(* Logix 5000 project; controller TWO_SRC_TEST vendor 1 type 14 code 54 rev 19.11; software revision 19.01 *)
// Two sources are connected to the same bus and power is shared between the two using a voltage droop controller.

TASK MainTask (continuous, watchdog 500 ms) : MainProgram

MODULES
   Local : vendor 1 type 14 code 54 (ICP 0, rev 19.11)
      CurrentMeasurement : 1756-IF8 (ICP 2, rev 1.1, Input RPI 100 ms)
      VoltageSetpoints : 1756-OF4 (ICP 1, rev 1.1, Output RPI 12 ms)
END_MODULES

VAR_GLOBAL   (* controller tags *)
   SOURCE_1_ControlSignal : ALIAS FOR Local:1:O.Ch0Data;
   SOURCE_1_Current : ALIAS FOR Local:2:I.Ch0Data;
   SOURCE_2_ControlSignal : ALIAS FOR Local:1:O.Ch1Data;
   SOURCE_2_Current : ALIAS FOR Local:2:I.Ch1Data;
END_VAR

PROGRAM MainProgram   (* main routine MainRoutine *)
VAR
   CURRENT_SCALING_FACTOR : REAL; {constant}
   MeasAddress : DINT;
   MeasArray : COUNTER;
   MeasCount : COUNTER;
   MeasCounter : COUNTER;
   MeasTimer : TIMER := (PRE := 10);
   NO_TRIM_CONTROL_SIGNAL : REAL := 1.23; {constant}
   SOURCE_1_CB : REAL[10];
   SOURCE_1_CurrentAverage : REAL;
   SOURCE_1_CurrentBuffer : REAL;
   SOURCE_1_DeltaV : REAL;
   SOURCE_1_DroopCoefficient : REAL;
   SOURCE_1_FullLoadCurrent : REAL;
   SOURCE_1_FullLoadVoltage : REAL;
   SOURCE_1_MAX_CONTROL_SIGNAL : REAL; {constant}
   SOURCE_1_MIN_CONTROL_SIGNAL : REAL; {constant}
   SOURCE_1_NoLoadVoltage : REAL;
   SOURCE_1_NominalVoltage : REAL; {constant}
   SOURCE_1_OutputVoltage : REAL;
   SOURCE_1_VoltageAdjustment : REAL;
   SOURCE_2_CB : REAL[10];
   SOURCE_2_CurrentAverage : REAL;
END_VAR

ROUTINE MainRoutine   (* ladder *)
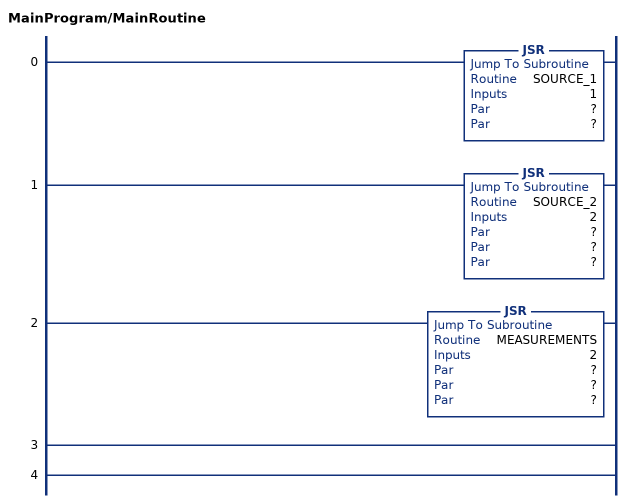
   0: JSR(SOURCE_1,1,?,?);
   1: JSR(SOURCE_2,2,?,?,?);
   2: JSR(MEASUREMENTS,2,?,?,?);
   3: ;
   4: ;
END_ROUTINE

ROUTINE MEASUREMENTS   (* ladder *)
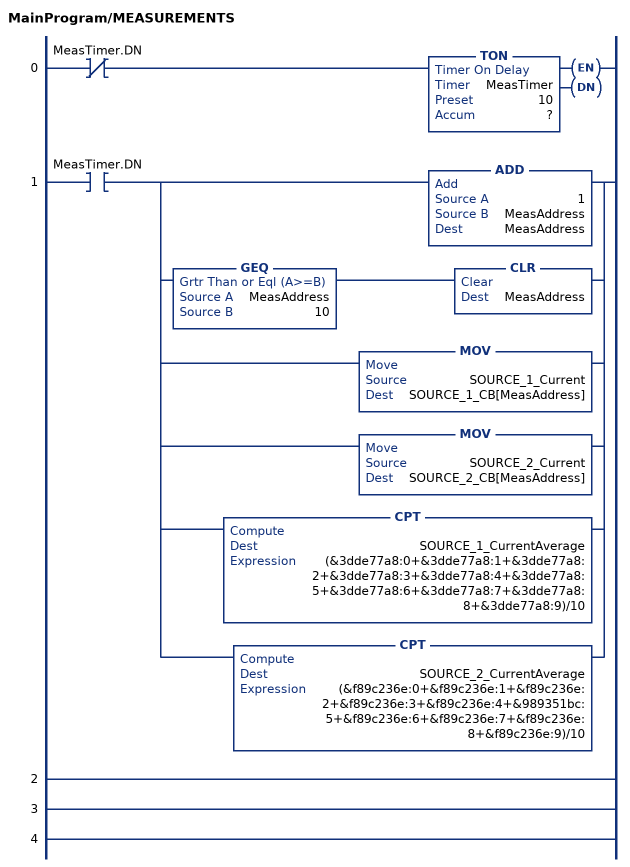
   0: XIO(MeasTimer.DN)TON(MeasTimer,?,?);
   1: XIC(MeasTimer.DN)[ADD(1,MeasAddress,MeasAddress) ,GEQ(MeasAddress,10) CLR(MeasAddress) ,MOV(SOURCE_1_Current,SOURCE_1_CB[MeasAddress]) ,MOV(SOURCE_2_Current,SOURCE_2_CB[MeasAddress]) ,CPT(SOURCE_1_CurrentAverage,(&3dde77a8:0+&3dde77a8:1+&3dde77a8:2+&3dde77a8:3+&3dde77a8:4+&3dde77a8:5+&3dde77a8:6+&3dde77a8:7+&3dde77a8:8+&3dde77a8:9)/10) ,CPT(SOURCE_2_CurrentAverage,(&f89c236e:0+&f89c236e:1+&f89c236e:2+&f89c236e:3+&f89c236e:4+&989351bc:5+&f89c236e:6+&f89c236e:7+&f89c236e:8+&f89c236e:9)/10) ];
   2: ;
   3: ;
   4: ;
END_ROUTINE

ROUTINE SOURCE_1   (* ladder *)
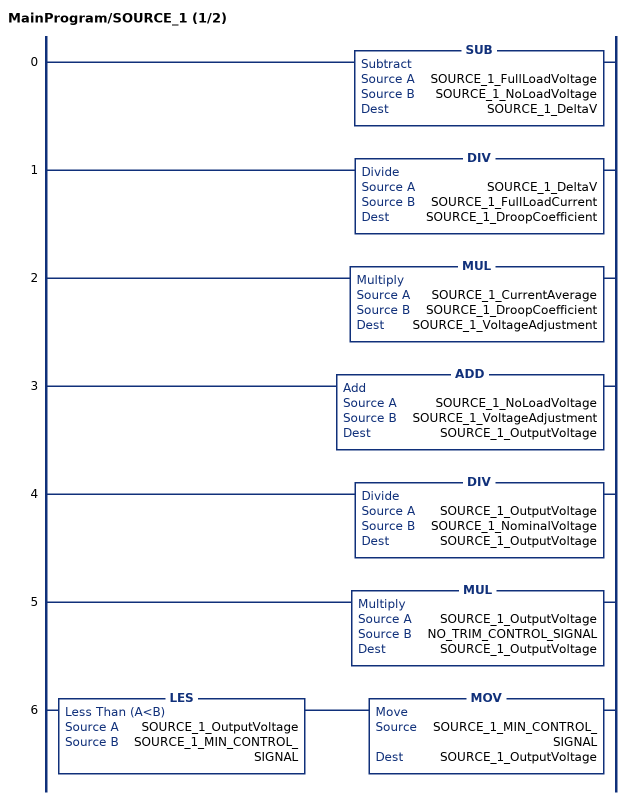
   0: SUB(SOURCE_1_FullLoadVoltage,SOURCE_1_NoLoadVoltage,SOURCE_1_DeltaV);
   1: DIV(SOURCE_1_DeltaV,SOURCE_1_FullLoadCurrent,SOURCE_1_DroopCoefficient);
   2: MUL(SOURCE_1_CurrentAverage,SOURCE_1_DroopCoefficient,SOURCE_1_VoltageAdjustment);
   3: ADD(SOURCE_1_NoLoadVoltage,SOURCE_1_VoltageAdjustment,SOURCE_1_OutputVoltage);
   4: DIV(SOURCE_1_OutputVoltage,SOURCE_1_NominalVoltage,SOURCE_1_OutputVoltage);
   5: MUL(SOURCE_1_OutputVoltage,NO_TRIM_CONTROL_SIGNAL,SOURCE_1_OutputVoltage);
   6: LES(SOURCE_1_OutputVoltage,SOURCE_1_MIN_CONTROL_SIGNAL)MOV(SOURCE_1_MIN_CONTROL_SIGNAL,SOURCE_1_OutputVoltage);
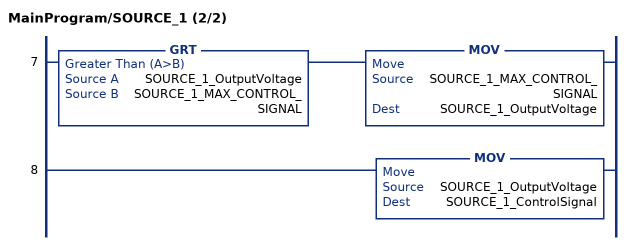
   7: GRT(SOURCE_1_OutputVoltage,SOURCE_1_MAX_CONTROL_SIGNAL)MOV(SOURCE_1_MAX_CONTROL_SIGNAL,SOURCE_1_OutputVoltage);
   8: MOV(SOURCE_1_OutputVoltage,SOURCE_1_ControlSignal);
END_ROUTINE
END_PROGRAM
